FUNCTION_BLOCK E_SPLIT_3 (* Split an event (generic FB) *)
  (* Standard: 61499-1 Annex A; Classification: event function block; Function: Split one event into two events; Description: Copyright (c) 2017, 2025 fortiss GmbH, HR Agrartechnik GmbH This program and the accompanying materials are made available under the terms of the Eclipse Public License 2.0 which is available at https://www.eclipse.org/legal/epl-2.0/ SPDX-License-Identifier: EPL-2.0 *)
  (* Version 3.0, 2025-04-14, Patrick Aigner, changed package *)
  (* Version 1.0.1, 2025-02-12, Franz Höpfinger, HR Agrartechnik GmbH, copy from E_SPLIT and make a E_SPLIT3 in the same way *)
  (* Version 1.0, 2017, Alois Zoitl, fortiss GmbH, initial API and implementation and/or initial documentation *)
  PACKAGE iec61499::events;
  {SET_ATTRIBUTE(eclipse4diac::core::GenericClassName, 'GEN_E_SPLIT')}
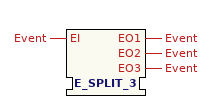
  EVENT_INPUT
    EI; (* Input event *)
  END_EVENT
  EVENT_OUTPUT
    EO1; (* First output event *)
    EO2; (* Second output event *)
    EO3;
  END_EVENT
END_FUNCTION_BLOCK
